PROGRAM My_Program
VAR
END_VAR

END_PROGRAM

(* stored: Version 1.1.0.1, ProductVersion 3.1.4024.16
   POU My_Program: Id {0a423137-b916-4f33-8548-42aef392f727}, SpecialFunc None *)
